# EPICS autosave request: iocBoot/ioc13idd_pg4/auto_settings.req
file "spinnaker_settings.req",            P=$(P),  R=cam1:
file "NDStdArrays_settings.req",          P=$(P),  R=image1:
file "commonPlugin_settings.req",         P=$(P)
$(P)cam1:GC_OnBoaColProEna
$(P)cam1:GC_VideoMode
